# EPICS autosave request: xx_auto_swait_settings.req
$(P)$(S).DESC
$(P)$(S).INAN
$(P)$(S).INBN
$(P)$(S).INCN
$(P)$(S).INDN
$(P)$(S).INEN
$(P)$(S).INFN
$(P)$(S).INGN
$(P)$(S).INHN
$(P)$(S).ININ
$(P)$(S).INJN
$(P)$(S).INKN
$(P)$(S).INLN
$(P)$(S).INAP
$(P)$(S).INBP
$(P)$(S).INCP
$(P)$(S).INDP
$(P)$(S).INEP
$(P)$(S).INFP
$(P)$(S).INGP
$(P)$(S).INHP
$(P)$(S).INIP
$(P)$(S).INJP
$(P)$(S).INKP
$(P)$(S).INLP
$(P)$(S).CALC
$(P)$(S).OUTN
$(P)$(S).OOPT
$(P)$(S).DOPT
$(P)$(S).DOLN
$(P)$(S).SCAN
$(P)$(S).ODLY
$(P)$(S).PREC
$(P)$(S).OEVT
